(* Logix 5000 project; controller MIXER Emulate 5570 rev 19.11; software revision 19.01 *)

TASK MainTask (continuous, watchdog 500 ms) : MainProgram

MODULES
   Local : Emulate 5570 (ICP 2, rev 19.11)
      IO : vendor 1 type 0 code 15 (ICP 3, rev 1.1, Output RPI 85 ms)
END_MODULES

VAR_GLOBAL   (* controller tags *)
   A : ALIAS FOR Local:3:O.Data[0].8;   // ALARMA
   ES : ALIAS FOR Local:3:O.Data[0].7;   // ESCANER
   L1 : ALIAS FOR Local:3:O.Data[0].3;   // LUZ ROJA
   L2 : ALIAS FOR Local:3:O.Data[0].4;   // LUZ AMARILLA
   L3 : ALIAS FOR Local:3:O.Data[0].5;   // LUZ VERDE
   M1 : ALIAS FOR Local:3:O.Data[0].1;   // ABRIR PUERTA
   M2 : ALIAS FOR Local:3:O.Data[0].2;   // CERRAR PUERTA
   ME : ALIAS FOR Local:3:O.Data[0].9;   // MENSAJE DE ESTADO
   MEN : STRING := 'SALDO INSUFICIENTE';   // MENSAJE 2
   P1 : ALIAS FOR Local:3:O.Data[0].6;   // PANTALLA DE ESTADO
   S1 : ALIAS FOR Local:3:I.Data[1].1;   // SENSOR DE AUTO
   S2 : ALIAS FOR Local:3:I.Data[1].2;   // SENSOR DE TARJETA DE ESCANER
   S3 : ALIAS FOR Local:3:I.Data[1].3;   // SENSOR DE SALDO DE TARJETA
   S4 : ALIAS FOR Local:3:I.Data[1].4;   // SENSOR LIMITE APERTURA PUERTA
   S5 : ALIAS FOR Local:3:I.Data[1].5;   // SENSOR LIMITE CERRADO PUERTA
   timer_01 : FBD_TIMER;
   timer_abrir : FBD_TIMER;
   timer_moroso : FBD_TIMER;
END_VAR

PROGRAM MainProgram   (* main routine MainRoutine *)
VAR
   Action_000 : SFC_ACTION := (Status := 16#0020_0000, PauseTimer := 1);
   Action_001 : SFC_ACTION := (Status := 16#0020_0000, PauseTimer := 1);
   Action_002 : SFC_ACTION := (Status := 16#0020_0000, PauseTimer := 1);
   Action_003 : SFC_ACTION := (Status := 16#0020_0000, PauseTimer := 1);
   Action_004 : SFC_ACTION := (Status := 16#0020_0000, PauseTimer := 1);
   Action_005 : SFC_ACTION := (Status := 16#0020_0000, PauseTimer := 1);
   Action_006 : SFC_ACTION := (Status := 16#0020_0000, PauseTimer := 1);
   Action_007 : SFC_ACTION := (Status := 16#0020_0000, PauseTimer := 1);
   Action_008 : SFC_ACTION := (Status := 16#0020_0000, PauseTimer := 1, T := 5000);
   Action_009 : SFC_ACTION := (Status := 16#0020_0000, PauseTimer := 1);
   Action_010 : SFC_ACTION := (Status := 16#0020_0000, PauseTimer := 1, T := 15000);
   DIST : DINT;
   ME1 : STRING := 'HELLO1';
   ME2 : STRING := 'HELLO2';
   PUERTA : DINT := 100;
   SENSOR_SALDO : DINT;
   SENSOR_TARJETA : DINT;
   Step_000 : SFC_STEP := (Status := 16#0020_0000, PauseTimer := 1);
   Step_001 : SFC_STEP := (Status := 16#0020_0000, PauseTimer := 1);
   Step_002 : SFC_STEP := (Status := 16#0020_0000, PauseTimer := 1);
   Step_003 : SFC_STEP := (Status := 16#0020_0000, PauseTimer := 1);
   Step_004 : SFC_STEP := (Status := 16#0020_0000, PauseTimer := 1);
   Step_005 : SFC_STEP := (Status := 16#0020_0000, PauseTimer := 1);
   Step_006 : SFC_STEP := (Status := 16#0020_0000, PauseTimer := 1);
   Step_007 : SFC_STEP := (Status := 16#0020_0000, PauseTimer := 1);
   Step_008 : SFC_STEP := (Status := 16#0020_0000, PauseTimer := 1);
   Step_009 : SFC_STEP := (Status := 16#0020_0000, PauseTimer := 1);
   Step_010 : SFC_STEP := (Status := 16#0020_0000, PauseTimer := 1);
   TEMPORARY : DINT;
   TIMER_PUERTA_ABRIR : TIMER := (PRE := 5000, ACC := 5010, EN := 1, DN := 1);
   TIMER_PUERTA_CERRAR : TIMER := (PRE := 5000);
   Tran_000 : BOOL;
   Tran_001 : BOOL;
   Tran_002 : BOOL;
   Tran_003 : BOOL;
   Tran_004 : BOOL;
   Tran_005 : BOOL;
   Tran_006 : BOOL;
   Tran_007 : BOOL;
   Tran_008 : BOOL;
   Tran_009 : BOOL;
   Tran_010 : BOOL;
END_VAR

ROUTINE MainRoutine   (* ladder *)
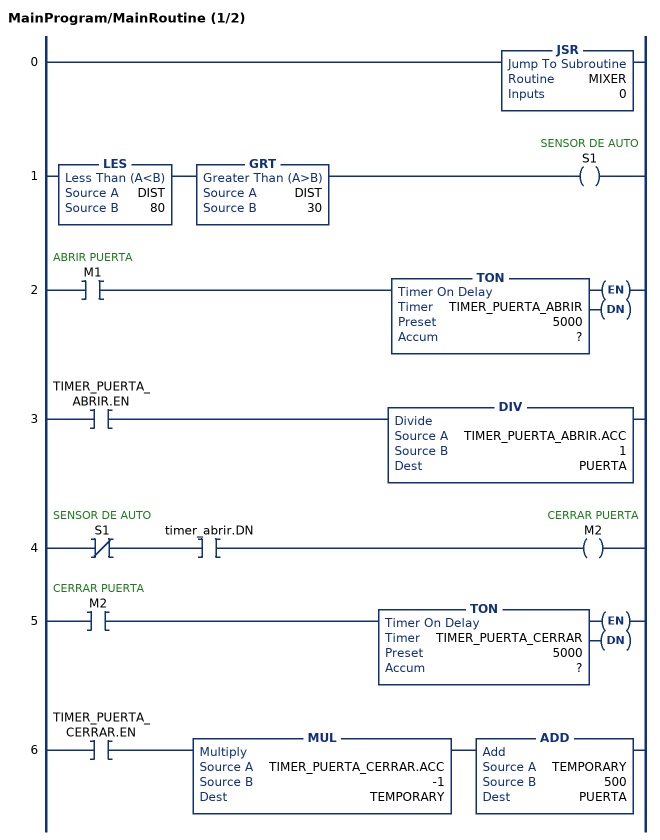
   0: JSR(MIXER,0);
   1: LES(DIST,80)GRT(DIST,30)OTE(S1);
   2: XIC(M1)TON(TIMER_PUERTA_ABRIR,?,?);
   3: XIC(TIMER_PUERTA_ABRIR.EN)DIV(TIMER_PUERTA_ABRIR.ACC,1,PUERTA);
   4: XIO(S1)XIC(timer_abrir.DN)OTE(M2);
   5: XIC(M2)TON(TIMER_PUERTA_CERRAR,?,?);
   6: XIC(TIMER_PUERTA_CERRAR.EN)MUL(TIMER_PUERTA_CERRAR.ACC,-1,TEMPORARY)ADD(TEMPORARY,500,PUERTA);
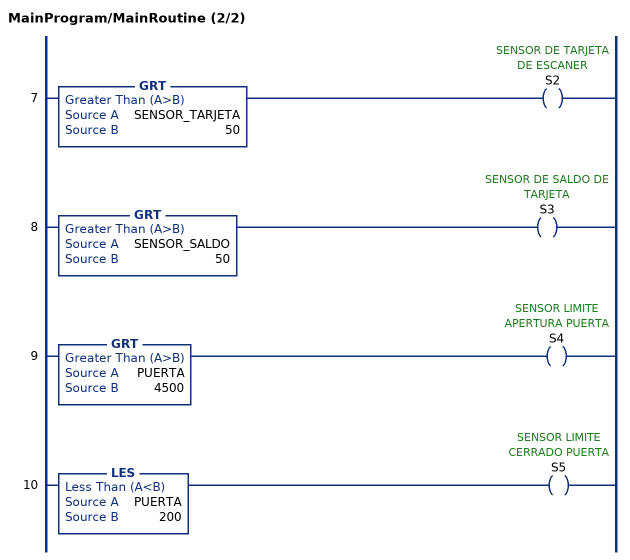
   7: GRT(SENSOR_TARJETA,50)OTE(S2);
   8: GRT(SENSOR_SALDO,50)OTE(S3);
   9: GRT(PUERTA,4500)OTE(S4);
   10: LES(PUERTA,200)OTE(S5);
END_ROUTINE

ROUTINE MIXER   (* sequential function chart *)
// SEMESTRAL
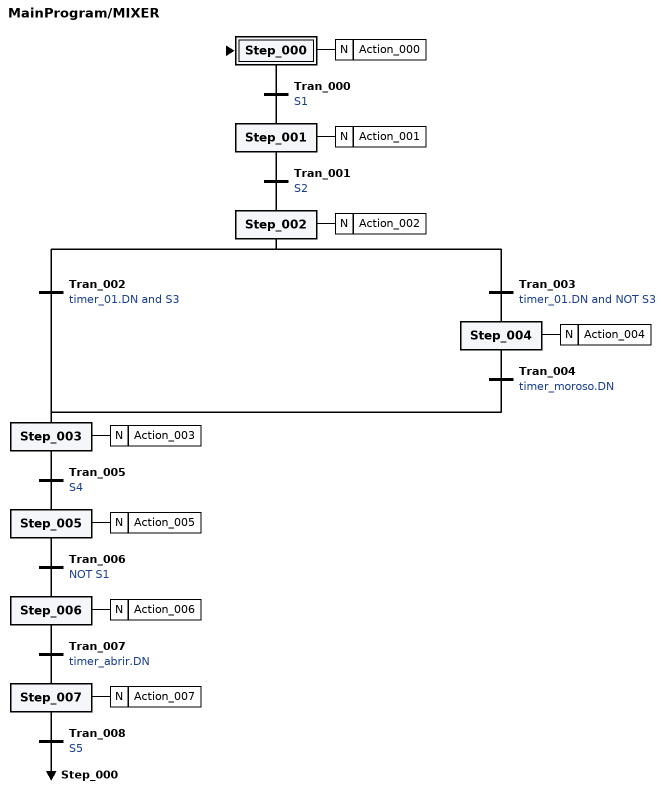
   INITIAL_STEP Step_000:
      ACTION Action_000 (N):
         M1:=0;M2:=0;L1:=0;L2:=0;L3:=0;
         P1:=0;ES:=0;
      END_ACTION
   END_STEP
   TRANSITION Tran_000 FROM Step_000 TO Step_001
      := S1
   END_TRANSITION
   STEP Step_001:
      ACTION Action_001 (N):
         P1:=0;L1:=0;L2:=1;L3:=0;
         ES:=1;
      END_ACTION
   END_STEP
   TRANSITION Tran_001 FROM Step_001 TO Step_002
      := S2
   END_TRANSITION
   STEP Step_002:
      ACTION Action_002 (N):
         L1:=0;L2:=1;L3:=0;
         timer_01.TimerEnable [:=] 1;
         TONR(timer_01);
         timer_01.Pre :=7000;
      END_ACTION
   END_STEP
   TRANSITION Tran_002 FROM Step_002 TO Step_003
      := timer_01.DN and S3
   END_TRANSITION
   TRANSITION Tran_003 FROM Step_002 TO Step_004
      := timer_01.DN and NOT S3
   END_TRANSITION
   STEP Step_004:
      ACTION Action_004 (N):
         ES:=0;A:=1;L1:=1;
         L2:=0;L3:=0;P1:=1;
         timer_moroso.TimerEnable [:=] 1;
         TONR(timer_moroso);
         timer_moroso.Pre :=15000;
      END_ACTION
   END_STEP
   STEP Step_003:
      ACTION Action_003 (N):
         L1:=0;L2:=1;L3:=0;M1:=1;
         A:=0;ES:=0;
      END_ACTION
   END_STEP
   TRANSITION Tran_005 FROM Step_003 TO Step_005
      := S4
   END_TRANSITION
   TRANSITION Tran_004 FROM Step_004 TO Step_003
      := timer_moroso.DN
   END_TRANSITION
   STEP Step_005:
      ACTION Action_005 (N):
         L1:=0;L2:=0;L3:=1;M1:=0;
      END_ACTION
   END_STEP
   TRANSITION Tran_006 FROM Step_005 TO Step_006
      := NOT S1
   END_TRANSITION
   STEP Step_006:
      ACTION Action_006 (N):
         timer_abrir.TimerEnable [:=] 1;
         TONR(timer_abrir);
         timer_abrir.Pre :=5000;
      END_ACTION
   END_STEP
   TRANSITION Tran_007 FROM Step_006 TO Step_007
      := timer_abrir.DN
   END_TRANSITION
   STEP Step_007:
      ACTION Action_007 (N):
         M2:=1;L1:=1;L2:=0;L3:=0;
      END_ACTION
   END_STEP
   TRANSITION Tran_008 FROM Step_007 TO Step_000
      := S5
   END_TRANSITION
END_ROUTINE
END_PROGRAM
